# EPICS autosave request: motorApp/Db/pseudoMotor_settings.req
# FILE... pseudoMotor_settings.req
$(P)$(M).DHLM
$(P)$(M).DLLM
$(P)$(M).TWV
$(P)$(M).DISA
$(P)$(M).DISP
$(P)$(M).OFF
$(P)$(M).VELO
$(P)$(M)C1
$(P)$(M)C2
$(P)$(M)C3
$(P)$(M)C4
$(P)$(M)C5
$(P)$(M)_able.VAL
$(P)$(M):scanParms.SP
$(P)$(M):scanParms.EP
$(P)$(M):scanParms.NP
